(* IEC 61131-3 sources: teller/JD_Teller_LC2_V11/Class/Write1, 1 file *)

(* ---- Write1.st ---- *)
(*!
<Class
	Name               = "Write1"
	Revision           = "0.0"
	RealtimeTask       = "false"
	CyclicTask         = "false"
	BackgroundTask     = "false"
	Sigmatek           = "false"
	OSInterface        = "false"
	HighPriority       = "false"
	Automatic          = "false"
	UpdateMode         = "Prescan"
	SharedCommandTable = "true"
	Objectsize         = "(284,120)">
	<Channels>
		<Server Name="ClassSvr" Visualized="false" Initialize="false" WriteProtected="true" Retentive="false"/>
		<Client Name="cWrite1" Required="true" Internal="false"/>
	</Channels>
</Class>
*)
Write1 : CLASS
  //Servers:
	ClassSvr 	: SvrChCmd_DINT;
  //Clients:
	cWrite1 	: CltCh_DINT;
  //Variables:
  //Functions:

	FUNCTION VIRTUAL GLOBAL Init;
  //Tables:
	FUNCTION @STD
		VAR_OUTPUT
			ret_code	: CONFSTATES;
		END_VAR;
	FUNCTION GLOBAL TAB @CT_;
END_CLASS;

FUNCTION VIRTUAL GLOBAL Write1::Init

  if    _FirstScan then
        cWrite1.Write (1);

  end_if;

END_FUNCTION
